// Mitsubishi GX Works2 project: BookEX6_44 Clock   PLC: Q13UDV

// global labels: Global
VAR_GLOBAL
  bVar0 AT M5000 : BOOL;
  abArray0 AT M5010 : ARRAY [0..49] OF BOOL;
  sStr0 AT D5000 : STRING[199];
  sStr1 AT D5100 : STRING[199];
  sStr2 AT D5200 : STRING[199];
  sStr3 AT D5300 : STRING[199];
  sStr4 AT D5400 : STRING[199];
  sStr5 AT D5500 : STRING[199];
  sStr6 AT D5600 : STRING[199];
  sStr7 AT D5700 : STRING[199];
  sStr8 AT D5800 : STRING[199];
  sStr9 AT D5900 : STRING[199];
  iVar0 AT D4500 : INT;
  iVar1 AT D4501 : INT;
  iVar2 AT D4502 : INT;
  iVar3 AT D4503 : INT;
  iVar4 AT D4504 : INT;
  iVar5 AT D4505 : INT;
  iVar6 AT D4506 : INT;
  iVar7 AT D4507 : INT;
  iVar8 AT D4508 : INT;
  iVar9 AT D4509 : INT;
  dVar0 AT D4510 : DINT;
  dVar1 AT D4512 : DINT;
  dVar2 AT D4514 : DINT;
  dVar3 AT D4516 : DINT;
  dVar4 AT D4518 : DINT;
  dVar5 AT D4520 : DINT;
  dVar6 AT D4522 : DINT;
  dVar7 AT D4524 : DINT;
  dVar8 AT D4526 : DINT;
  dVar9 AT D4528 : DINT;
  wVar0 AT D4530 : WORD;
  wVar1 AT D4531 : WORD;
  wVar2 AT D4532 : WORD;
  wVar3 AT D4533 : WORD;
  wVar4 AT D4534 : WORD;
  wVar5 AT D4535 : WORD;
  wVar6 AT D4536 : WORD;
  wVar7 AT D4537 : WORD;
  wVar8 AT D4538 : WORD;
  wVar9 AT D4539 : WORD;
  dwVar0 AT D4540 : DWORD;
  dwVar1 AT D4542 : DWORD;
  dwVar2 AT D4544 : DWORD;
  dwVar3 AT D4546 : DWORD;
  dwVar4 AT D4548 : DWORD;
  dwVar5 AT D4550 : DWORD;
  dwVar6 AT D4552 : DWORD;
  dwVar7 AT D4554 : DWORD;
  dwVar8 AT D4556 : DWORD;
  dwVar9 AT D4558 : DWORD;
  fsVar0 AT D4560 : REAL;
  fsVar1 AT D4562 : REAL;
  fsVar2 AT D4564 : REAL;
  fsVar3 AT D4566 : REAL;
  fsVar4 AT D4568 : REAL;
  fsVar5 AT D4570 : REAL;
  fsVar6 AT D4572 : REAL;
  fsVar7 AT D4574 : REAL;
  fsVar8 AT D4576 : REAL;
  fsVar9 AT D4578 : REAL;
  fdVar0 AT D4580 : LREAL;
  tTime0 AT D4620 : TIME;
  tTime1 AT D4622 : TIME;
  tTime2 AT D4624 : TIME;
  tTime3 AT D4626 : TIME;
  tTime4 AT D4628 : TIME;
  tTime5 AT D4630 : TIME;
  tTime6 AT D4632 : TIME;
  tTime7 AT D4634 : TIME;
  tTime8 AT D4636 : TIME;
  tTime9 AT D4638 : TIME;
  tTime10 AT D4640 : TIME;
  bVar1 AT M5001 : BOOL;
  bVar2 AT M5002 : BOOL;
  bVar3 AT M5003 : BOOL;
  bVar4 AT M5004 : BOOL;
  bVar5 AT M5005 : BOOL;
  bVar6 AT M5006 : BOOL;
  bVar7 AT M5007 : BOOL;
  bVar8 AT M5008 : BOOL;
  bVar9 AT M5009 : BOOL;
  abArray1 AT M5060 : ARRAY [0..49] OF BOOL;
  abArray2 AT M5110 : ARRAY [0..49] OF BOOL;
  abArray3 AT M5160 : ARRAY [0..49] OF BOOL;
  abArray4 AT M5210 : ARRAY [0..49] OF BOOL;
  abArray5 AT M5260 : ARRAY [0..49] OF BOOL;
  abArray6 AT M5310 : ARRAY [0..49] OF BOOL;
  abArray7 AT M5360 : ARRAY [0..49] OF BOOL;
  abArray8 AT M5410 : ARRAY [0..49] OF BOOL;
  abArray9 AT M5460 : ARRAY [0..49] OF BOOL;
  fdVar1 AT D4584 : LREAL;
  fdVar2 AT D4588 : LREAL;
  fdVar3 AT D4592 : LREAL;
  fdVar4 AT D4596 : LREAL;
  fdVar5 AT D4600 : LREAL;
  fdVar6 AT D4604 : LREAL;
  fdVar7 AT D4608 : LREAL;
  fdVar8 AT D4612 : LREAL;
  fdVar9 AT D4616 : LREAL;
  afsPen0 AT D2000 : ARRAY [0..499] OF REAL;
  afsPen1 AT D3000 : ARRAY [0..499] OF REAL;
  adwD10 AT D10 : ARRAY [0..9] OF DWORD;
  awD10 AT D10 : ARRAY [0..19] OF WORD;
  abM10 AT M10 : ARRAY [0..19] OF BOOL;
  bDown AT M50 : BOOL;
  bUp AT M51 : BOOL;
  bResult AT M325 : ARRAY [0..2] OF BOOL;
  bResultCMP1 AT M328 : ARRAY [0..2] OF BOOL;
  bResultCMP2 AT M331 : ARRAY [0..2] OF BOOL;
  bResultCP1 AT M334 : ARRAY [0..2] OF BOOL;
  bResultCP2 AT M337 : ARRAY [0..2] OF BOOL;
  aiClock AT D40 : ARRAY [0..6] OF INT;
  aiClock1 AT D40 : ARRAY [0..7] OF INT;
  aiClock2 AT D40 : ARRAY [0..5] OF INT;
  iInYear AT D48 : INT;
  iInMonth AT D49 : INT;
  asDay AT D100 : ARRAY [0..49] OF STRING[3] := [50('')];
  aiLowDate AT D330 : ARRAY [0..5] OF INT;
  aiLowTime AT D333 : ARRAY [0..2] OF INT;
  aiHighDate AT D340 : ARRAY [0..5] OF INT;
  aiHighTime AT D343 : ARRAY [0..2] OF INT;
  aiChkDate AT D350 : ARRAY [0..5] OF INT;
  aiChkTime AT D353 : ARRAY [0..2] OF INT;
  aiCnvTime AT D360 : ARRAY [0..2] OF INT;
  dCnvSec AT D363 : DINT;
END_VAR
// user libraries (not included): HMI

FUNCTION_BLOCK Calendar
VAR_INPUT
  i_Year : INT;
  i_Month : INT;
END_VAR
VAR
  oldYear : INT;
  oldMonth : INT;
  Days : INT;
  GetLastDay_1 : GetLastDay;
  ix : INT;
  iy : INT;
  iz : INT;
  sTemp : STRING[9];
  sForm : DINT;
  GetDayOfWeek_1 : GetDayOfWeek;
END_VAR
;

IF (oldMonth = i_Month) AND (oldYear = i_Year) THEN
	RETURN;
END_IF;

GetLastDay_1(bEN:= TRUE, iYear:= i_Year, iMonth:= i_Month );
Days := GetLastDay_1.o_LastDay;
GetDayOfWeek_1(bEN:=TRUE,iYear:= i_Year, iMonth:= i_Month, iDay:= 1);
iy :=  GetDayOfWeek_1.o_DayWeek;
iz := iy + Days;
sForm := 3;

FOR ix := 0 TO 41 DO 
	IF ( ix >= iy ) AND ( ix < iz) THEN
		STR(TRUE, sForm, ix-iy+1, sTemp);
		sTemp := DELETE(sTemp, 1, 1); 
	ELSE
		sTemp := '';
	END_IF;	
	asDay[ix] := sTemp;
END_FOR;

oldMonth := i_Month;
oldYear := i_Year;
END_FUNCTION_BLOCK

FUNCTION_BLOCK CmpDateZone
VAR_INPUT
  bEN : BOOL;
END_VAR
VAR_OUTPUT
  bENO : BOOL;
END_VAR
VAR_INPUT
  LowerLimit : ARRAY [0..5] OF INT;
  UpperLimit : ARRAY [0..5] OF INT;
  CheckDate : ARRAY [0..5] OF INT;
END_VAR
VAR_OUTPUT
  bLower : BOOL;
  bInner : BOOL;
  bUpper : BOOL;
END_VAR
VAR
  dLLimit : DINT;
  dULimit : DINT;
  dChkDate : DINT;
  bChkBit : ARRAY [0..2] OF BOOL;
  bChkData1 : BOOL;
  bChkData2 : BOOL;
  bChkData3 : BOOL;
END_VAR

bENO 	:= bEN;
bChkBit[0]	:= FALSE;
bChkBit[1]	:= FALSE;
bChkBit[2]	:= FALSE;
bChkData1 := (CheckDate[0]<2000) OR (CheckDate[0]>2067) 
  	OR (CheckDate[1]=0) OR (CheckDate[1]>12) 
  	OR (CheckDate[2]=0) OR (CheckDate[2]>31)  
  	OR (CheckDate[3]>23) OR (CheckDate[4]>59) OR (CheckDate[5]>59);
bChkData2 := (LowerLimit[0]<2000) OR (LowerLimit[0]>2067) 
  	OR (LowerLimit[1]=0) OR (LowerLimit[1]>12) 
  	OR (LowerLimit[2]=0) OR (LowerLimit[2]>31)  
  	OR (LowerLimit[3]>23) OR (LowerLimit[4]>59) OR (LowerLimit[5]>59);
bChkData3 := (UpperLimit[0]<2000) OR (UpperLimit[0]>2067) 
  	OR (UpperLimit[1]=0) OR (UpperLimit[1]>12) 
  	OR (UpperLimit[2]=0) OR (UpperLimit[2]>31)  
  	OR (UpperLimit[3]>23) OR (UpperLimit[4]>59) OR (UpperLimit[5]>59);
  		  		 
IF NOT bEN OR bChkData1 OR bChkData2 OR bChkData3 THEN
	RETURN;
END_IF; 
  
dLLimit := newDATE2SEC(LowerLimit[0], LowerLimit[1], LowerLimit[2], LowerLimit[3], LowerLimit[4], LowerLimit[5]);
dULimit := newDATE2SEC(UpperLimit[0], UpperLimit[1],UpperLimit[2],UpperLimit[3],UpperLimit[4],UpperLimit[5]); 
dChkDate := newDATE2SEC(CheckDate[0], CheckDate[1],CheckDate[2],CheckDate[3],CheckDate[4],CheckDate[5]);
IF dLLimit > dChkDate THEN
	bChkBit[0] := TRUE;
ELSIF dULimit < dChkDate THEN	
	bChkBit[2] := TRUE;
ELSE
	bChkBit[1] := TRUE;
END_IF;
bLower	:= bChkBit[0];
bUpper	:= bChkBit[2];
bInner	:= bChkBit[1];
END_FUNCTION_BLOCK

FUNCTION_BLOCK GetDayOfWeek
VAR_INPUT
  bEN : BOOL;
END_VAR
VAR_OUTPUT
  bENO : BOOL;
END_VAR
VAR_INPUT
  iYear : INT;
END_VAR
VAR_OUTPUT
  o_DayWeek : INT;
END_VAR
VAR
  Result : INT;
END_VAR
VAR_INPUT
  iMonth : INT;
  iDay : INT;
END_VAR
VAR
  iY : INT;
  iC : INT;
  iM : INT;
  iYear2 : INT;
END_VAR

bENO 	:= bEN;
IF NOT bEN THEN
	RETURN;
END_IF;
IF iMonth <= 2 THEN
	iYear2 := iYear - 1;
	iM := iMonth + 12;
ELSE
	iYear2 := iYear;
	iM := iMonth;
END_IF;
iC := iYear2 / 100; 
iY := iYear2 MOD 100;
Result := ( (21*iC)/4 +(5* iY)/4 + (13 * (iM+1)) / 5 +iDay - 1) MOD 7; 
o_DayWeek := Result;
END_FUNCTION_BLOCK

FUNCTION_BLOCK GetLastDay
VAR_INPUT
  bEN : BOOL;
END_VAR
VAR_OUTPUT
  bENO : BOOL;
END_VAR
VAR_INPUT
  iYear : INT;
END_VAR
VAR_OUTPUT
  o_LastDay : INT;
END_VAR
VAR
  Result : INT;
END_VAR
VAR_INPUT
  iMonth : INT;
END_VAR
VAR
  bLeap : BOOL;
END_VAR

bENO 	:= bEN;
IF NOT bEN THEN
	RETURN;
END_IF; 

bLeap := LeapYear(iYear);
CASE iMonth OF
	1 : Result	:= 31;
	2 : IF bLeap THEN Result := 29; ELSE Result	:= 28; END_IF;
	3 : Result	:= 31;
	4 : Result	:= 30;
	5 : Result	:= 31;
	6 : Result	:= 30;
	7 : Result	:= 31;
	8 : Result	:= 31;
	9 : Result	:= 30;
	10 : Result	:= 31;
	11 : Result	:= 30;
	12 : Result	:= 31;
END_CASE;	
o_LastDay := Result;
END_FUNCTION_BLOCK

FUNCTION_BLOCK HourMeter
VAR_INPUT
  bEN : BOOL;
END_VAR
VAR_OUTPUT
  bENO : BOOL;
END_VAR
VAR_INPUT
  iHour : INT;
  iCurrHour : INT;
  iCurrSec : INT;
END_VAR
VAR_OUTPUT
  etHour : INT;
  etSec : INT;
  bOut : BOOL;
END_VAR
VAR
  tmpHour : INT;
  tmpSec : INT;
  R_TRIG_1 : R_TRIG;
END_VAR

bENO 	:= bEN;
IF LDP(TRUE, bEN) THEN
	tmpHour	:= iCurrHour;
	tmpSec	:= iCurrSec;
	bOut	:= FALSE;
END_IF;
IF NOT bEN THEN
	RETURN;
END_IF; 


IF LDP(TRUE, SM412) THEN
	tmpSec	:= tmpSec+1;
	IF tmpSec > 3599 THEN
		tmpSec	:= 0;
		tmpHour	:= tmpHour+1;
	END_IF;
	IF tmpHour = iHour THEN
		bOut	:= TRUE;
	END_IF;
END_IF;

etHour	:= tmpHour;
etSec	:= tmpSec;
END_FUNCTION_BLOCK

FUNCTION LeapYear
VAR
  bLeap4 : BOOL;
  bLeap100 : BOOL;
  bLeap400 : BOOL;
END_VAR
VAR_INPUT
  i_Year : INT;
END_VAR
VAR
  bLeap : BOOL;
END_VAR
;
bLeap := FALSE;
IF (i_Year MOD 4) = 0 THEN bLeap4 := TRUE; ELSE bLeap4 := FALSE; END_IF;
IF (i_Year MOD 100) = 0 THEN bLeap100 := TRUE; ELSE bLeap100 := FALSE; END_IF;
IF (i_Year MOD 400) = 0 THEN bLeap400 := TRUE; ELSE bLeap400 := FALSE; END_IF;
IF (bLeap4 AND NOT bLeap100) OR bLeap400 THEN bLeap := TRUE; END_IF;
LeapYear := bLeap;
END_FUNCTION

FUNCTION newDATE2SEC
VAR_INPUT
  i_Year : INT;
  i_Month : INT;
  i_Day : INT;
  i_Hour : INT;
  i_Min : INT;
  i_Sec : INT;
END_VAR
VAR
  ix : INT;
  dDay : DINT;
  diDay : DINT;
END_VAR
;
IF i_Year  < 2000  OR i_Year > 2067 THEN 
	newDATE2SEC := 0;
	RETURN;
END_IF; 
dDay := 0;
IF i_Year > 2000 THEN
	FOR ix := 2000 TO i_Year-1 DO 
		IF LeapYear(ix) THEN
			dDay := dDay + 366;
		ELSE
			dDay := dDay + 365;
		END_IF;
	END_FOR;
END_IF;
diDay := INT_TO_DINT(i_Day-1);
CASE i_Month OF
	1 : 	dDay := dDay + diDay;
	2 :	dDay := dDay + 31 + diDay;
	3 : 	dDay := dDay + 31 + 28 + diDay;
	4 : 	dDay := dDay + 31 + 28 + 31 + diDay;
	5 : 	dDay := dDay + 31 + 28 + 31 + 30 + diDay;
	6 : 	dDay := dDay + 31 + 28 + 31 + 30 + 31 + diDay;
	7 : 	dDay := dDay + 31 + 28 + 31 + 30 + 31 + 30 + diDay;
	8 : 	dDay := dDay + 31 + 28 + 31 + 30 + 31 + 30 + 31 + diDay;
	9 : 	dDay := dDay + 31 + 28 + 31 + 30 + 31 + 30 + 31 + 31 + diDay;
	10 : 	dDay := dDay + 31 + 28 + 31 + 30 + 31 + 30 + 31 + 31 + 30 + diDay;
	11 : 	dDay := dDay + 31 + 28 + 31 + 30 + 31 + 30 + 31 + 31 + 30 + 31 + diDay;
	12 : 	dDay := dDay + 31 + 28 + 31 + 30 + 31 + 30 + 31 + 31 + 30 + 31 + 30 + diDay;
ELSE
	dDay := 0;
END_CASE;
IF i_Month > 2 AND LeapYear(i_Year) THEN dDay := dDay + 1; END_IF;
newDATE2SEC := dDay * 24* 60 * 60 + INT_TO_DINT(i_Hour) * 60 * 60 + INT_TO_DINT(i_Min) * 60 + INT_TO_DINT(i_Sec);
END_FUNCTION

FUNCTION_BLOCK sysDateTime
VAR_OUTPUT
  Secs : INT;
  Mins : INT;
  Hours : INT;
  Day : INT;
  Month : INT;
  Year : INT;
END_VAR
VAR
  Temp2 : WORD;
  Temp1 : WORD;
  fbTimer : TON;
  SeqGet : INT;
END_VAR
(* PLC의 realtime clock data를 읽는다 *)
SM213 := TRUE;
(* Year *)
Temp1 := SHR(INT_TO_WORD(SD210) AND 16#FF00, 8);
Temp2 := INT_TO_WORD(SD213) AND 16#FF00;
BIN(TRUE, Temp1 OR Temp2, Year);
(* Month *)
Temp1 := INT_TO_WORD(SD210) AND 16#00FF;
BIN(TRUE, Temp1, Month);
(* Day *)
Temp1 := SHR(INT_TO_WORD(SD211) AND 16#FF00, 8);
BIN(TRUE, Temp1, Day);
(* Hour *)
Temp1 := INT_TO_WORD(SD211) AND 16#00FF;
BIN(TRUE, Temp1, Hours);
(* Minute *)
Temp1 := SHR(INT_TO_WORD(SD212) AND 16#FF00, 8);
BIN(TRUE, Temp1, Mins);
(* Second *)
Temp1 := INT_TO_WORD(SD212) AND 16#00FF;
BIN(TRUE, Temp1, Secs);
END_FUNCTION_BLOCK

PROGRAM ExCalendar
VAR
  Calendar_1 : Calendar;
  aiMin : ARRAY [0..1] OF INT;
  aiSec : ARRAY [0..1] OF INT;
  aiHour : ARRAY [0..1] OF INT;
END_VAR
(* structured ladder/FBD written out as ST: instructions are called as NAME(EN, inputs, outputs); _pN, _eN, _tN stand for wires *)
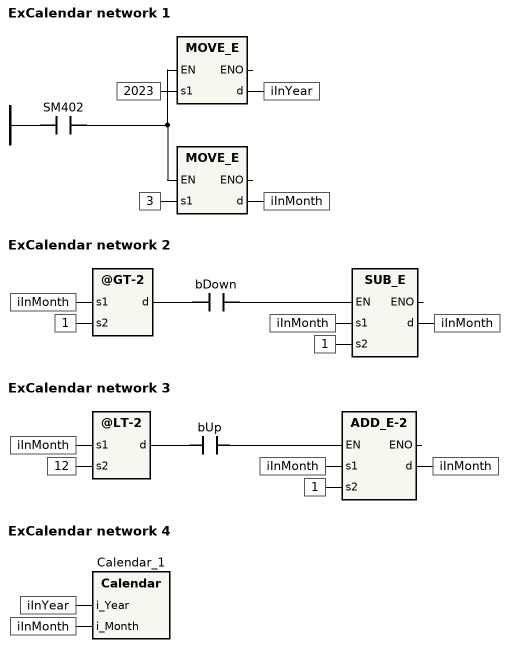
(* network 1 *)
MOVE_E(SM402, 2023, iInYear);
MOVE_E(SM402, 3, iInMonth);
(* network 2 *)
SUB_E(@GT-2(iInMonth, 1) AND bDown, iInMonth, 1, iInMonth);
(* network 3 *)
ADD_E(@LT-2(iInMonth, 12) AND bUp, iInMonth, 1, iInMonth);
(* network 4 *)
Calendar_1(i_Year := iInYear, i_Month := iInMonth);
END_PROGRAM

PROGRAM ExClcok
VAR
  Calendar_1 : Calendar;
  aiMin : ARRAY [0..1] OF INT;
  aiSec : ARRAY [0..1] OF INT;
  aiHour : ARRAY [0..1] OF INT;
END_VAR
(* structured ladder/FBD written out as ST: instructions are called as NAME(EN, inputs, outputs); _pN, _eN, _tN stand for wires *)
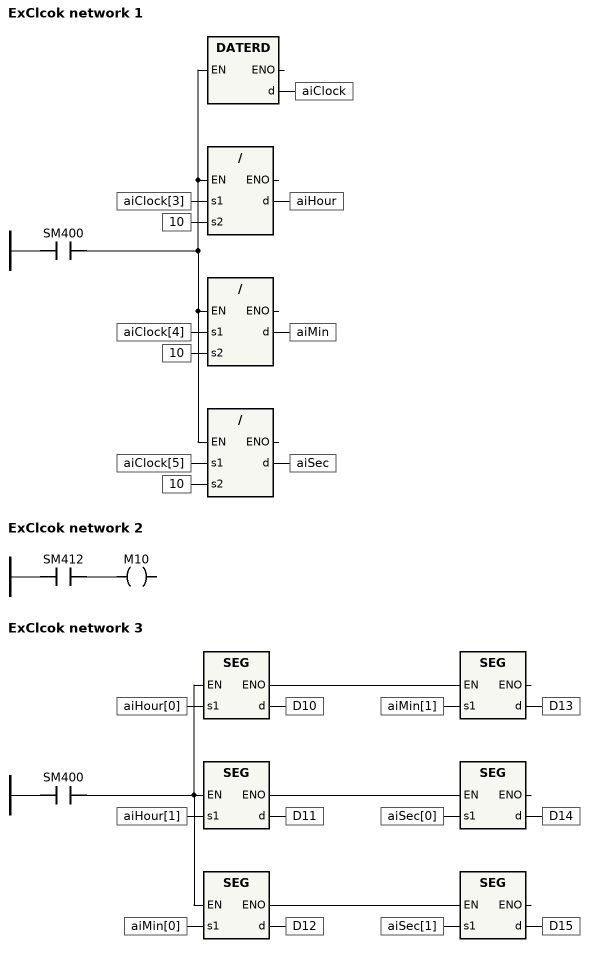
(* network 1 *)
DATERD(SM400, aiClock);
/(SM400, aiClock[3], 10, aiHour);
/(SM400, aiClock[4], 10, aiMin);
/(SM400, aiClock[5], 10, aiSec);
(* network 2 *)
M10 := SM412;
(* network 3 *)
_e1 := SEG(SM400, aiHour[0], D10);
SEG(_e1, aiMin[1], D13);
_e2 := SEG(SM400, aiHour[1], D11);
SEG(_e2, aiSec[0], D14);
_e3 := SEG(SM400, aiMin[0], D12);
SEG(_e3, aiSec[1], D15);
END_PROGRAM

PROGRAM ExDATE2SEC
VAR
  aiDate : ARRAY [0..5] OF INT;
END_VAR
(* structured ladder/FBD written out as ST: instructions are called as NAME(EN, inputs, outputs); _pN, _eN, _tN stand for wires *)
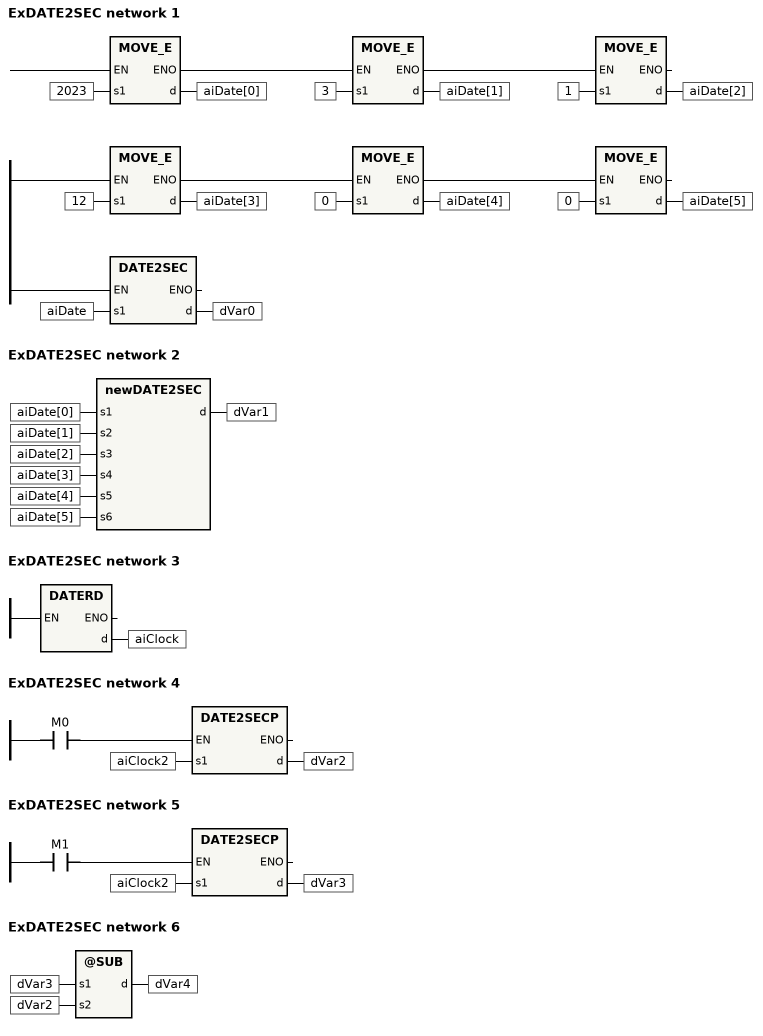
(* network 1 *)
_e1 := MOVE_E(TRUE, 2023, aiDate[0]);
_e2 := MOVE_E(_e1, 3, aiDate[1]);
MOVE_E(_e2, 1, aiDate[2]);
_e3 := MOVE_E(TRUE, 12, aiDate[3]);
_e4 := MOVE_E(_e3, 0, aiDate[4]);
MOVE_E(_e4, 0, aiDate[5]);
DATE2SEC(TRUE, aiDate, dVar0);
(* network 2 *)
dVar1 := newDATE2SEC(aiDate[0], aiDate[1], aiDate[2], aiDate[3], aiDate[4], aiDate[5]);
(* network 3 *)
DATERD(TRUE, aiClock);
(* network 4 *)
DATE2SECP(M0, aiClock2, dVar2);
(* network 5 *)
DATE2SECP(M1, aiClock2, dVar3);
(* network 6 *)
dVar4 := @SUB(dVar3, dVar2);
END_PROGRAM

PROGRAM ExDateMinus
VAR
  Mov4INT_3 : Mov4INT;
  Mov4INT_4 : Mov4INT;
  aiTime1 : ARRAY [0..2] OF INT;
  aiTime2 : ARRAY [0..2] OF INT;
  aiTime3 : ARRAY [0..2] OF INT;
  Mov4INT_1 : Mov4INT;
END_VAR
(* structured ladder/FBD written out as ST: instructions are called as NAME(EN, inputs, outputs); _pN, _eN, _tN stand for wires *)
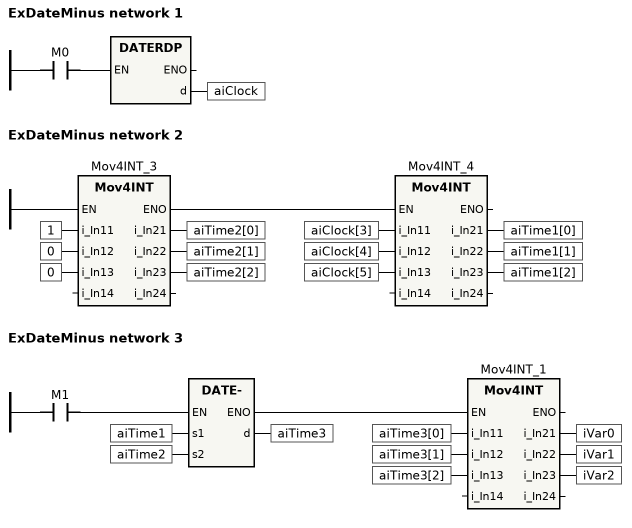
(* network 1 *)
DATERDP(M0, aiClock);
(* network 2 *)
Mov4INT_3(EN := TRUE, i_In11 := 1, i_In12 := 0, i_In13 := 0, i_In21 => aiTime2[0], i_In22 => aiTime2[1], i_In23 => aiTime2[2]);
Mov4INT_4(EN := Mov4INT_3.ENO, i_In11 := aiClock[3], i_In12 := aiClock[4], i_In13 := aiClock[5], i_In21 => aiTime1[0], i_In22 => aiTime1[1], i_In23 => aiTime1[2]);
(* network 3 *)
_e1 := DATE-(M1, aiTime1, aiTime2, aiTime3);
Mov4INT_1(EN := _e1, i_In11 := aiTime3[0], i_In12 := aiTime3[1], i_In13 := aiTime3[2], i_In21 => iVar0, i_In22 => iVar1, i_In23 => iVar2);
END_PROGRAM

PROGRAM ExDatePlus
VAR
  Mov4INT_3 : Mov4INT;
  Mov4INT_4 : Mov4INT;
  aiTime1 : ARRAY [0..2] OF INT;
  aiTime2 : ARRAY [0..2] OF INT;
  aiTime3 : ARRAY [0..2] OF INT;
  Mov4INT_1 : Mov4INT;
END_VAR
(* structured ladder/FBD written out as ST: instructions are called as NAME(EN, inputs, outputs); _pN, _eN, _tN stand for wires *)
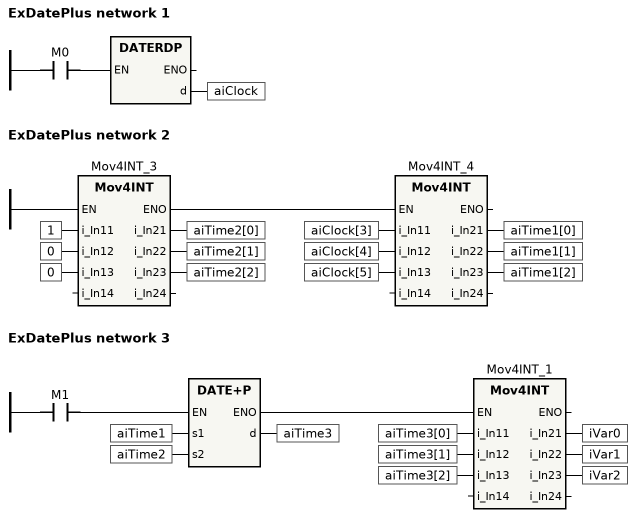
(* network 1 *)
DATERDP(M0, aiClock);
(* network 2 *)
Mov4INT_3(EN := TRUE, i_In11 := 1, i_In12 := 0, i_In13 := 0, i_In21 => aiTime2[0], i_In22 => aiTime2[1], i_In23 => aiTime2[2]);
Mov4INT_4(EN := Mov4INT_3.ENO, i_In11 := aiClock[3], i_In12 := aiClock[4], i_In13 := aiClock[5], i_In21 => aiTime1[0], i_In22 => aiTime1[1], i_In23 => aiTime1[2]);
(* network 3 *)
_e1 := DATE+P(M1, aiTime1, aiTime2, aiTime3);
Mov4INT_1(EN := _e1, i_In11 := aiTime3[0], i_In12 := aiTime3[1], i_In13 := aiTime3[2], i_In21 => iVar0, i_In22 => iVar1, i_In23 => iVar2);
END_PROGRAM

PROGRAM ExDATERD
VAR
  wBCD1 : WORD;
  wBCD2 : WORD;
  wBCD3 : WORD;
  wBCD4 : WORD;
  wBCD5 : WORD;
  wBCD6 : WORD;
  wBCD7 : WORD;
  wBCD8 : WORD;
  iTime1 : INT;
  iTime2 : INT;
  iTime3 : INT;
  iTime4 : INT;
  iTime5 : INT;
  iTime6 : INT;
  iTime7 : INT;
  iTime8 : INT;
  sysDateTime_1 : sysDateTime;
  Mov8INT2BCD_1 : Mov8INT2BCD;
END_VAR
(* structured ladder/FBD written out as ST: instructions are called as NAME(EN, inputs, outputs); _pN, _eN, _tN stand for wires *)
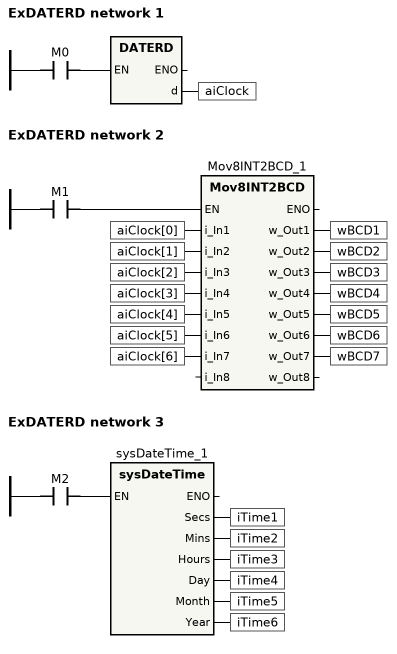
(* network 1 *)
DATERD(M0, aiClock);
(* network 2 *)
Mov8INT2BCD_1(EN := M1, i_In1 := aiClock[0], i_In2 := aiClock[1], i_In3 := aiClock[2], i_In4 := aiClock[3], i_In5 := aiClock[4], i_In6 := aiClock[5], i_In7 := aiClock[6], w_Out1 => wBCD1, w_Out2 => wBCD2, w_Out3 => wBCD3, w_Out4 => wBCD4, w_Out5 => wBCD5, w_Out6 => wBCD6, w_Out7 => wBCD7);
(* network 3 *)
sysDateTime_1(EN := M2, Secs => iTime1, Mins => iTime2, Hours => iTime3, Day => iTime4, Month => iTime5, Year => iTime6);
END_PROGRAM

PROGRAM ExDateWR
VAR
  acVar0 : ARRAY [0..6] OF INT;
END_VAR
(* structured ladder/FBD written out as ST: instructions are called as NAME(EN, inputs, outputs); _pN, _eN, _tN stand for wires *)
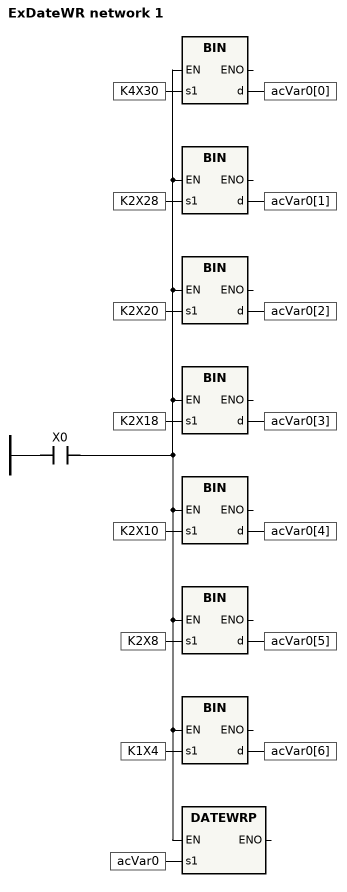
(* network 1 *)
BIN(X0, K4X30, acVar0[0]);
BIN(X0, K2X28, acVar0[1]);
BIN(X0, K2X20, acVar0[2]);
BIN(X0, K2X18, acVar0[3]);
BIN(X0, K2X10, acVar0[4]);
BIN(X0, K2X8, acVar0[5]);
BIN(X0, K1X4, acVar0[6]);
DATEWRP(X0, acVar0);
END_PROGRAM

PROGRAM ExGetLastDay
VAR
  GetLastDay_1 : GetLastDay;
  GetLastDay_2 : GetLastDay;
  GetLastDay_3 : GetLastDay;
  GetLastDay_4 : GetLastDay;
  GetLastDay_5 : GetLastDay;
  GetLastDay_6 : GetLastDay;
END_VAR
(* structured ladder/FBD written out as ST: instructions are called as NAME(EN, inputs, outputs); _pN, _eN, _tN stand for wires *)
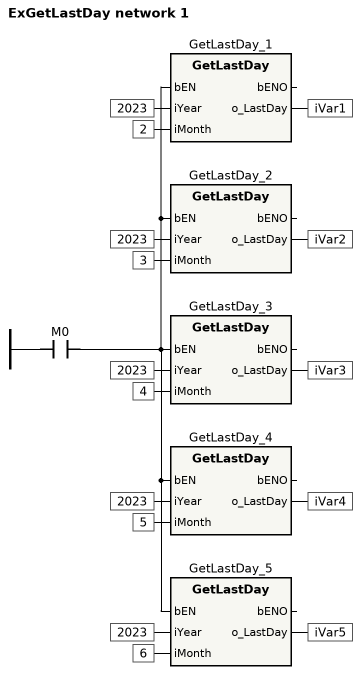
(* network 1 *)
GetLastDay_1(bEN := M0, iYear := 2023, iMonth := 2, o_LastDay => iVar1);
GetLastDay_2(bEN := M0, iYear := 2023, iMonth := 3, o_LastDay => iVar2);
GetLastDay_3(bEN := M0, iYear := 2023, iMonth := 4, o_LastDay => iVar3);
GetLastDay_4(bEN := M0, iYear := 2023, iMonth := 5, o_LastDay => iVar4);
GetLastDay_5(bEN := M0, iYear := 2023, iMonth := 6, o_LastDay => iVar5);
END_PROGRAM

PROGRAM ExHOUR
VAR
  aiVar3 : ARRAY [0..2] OF INT;
  iHourData : INT;
  iSecData : INT;
  aiVar4 : ARRAY [0..2] OF INT;
END_VAR
(* structured ladder/FBD written out as ST: instructions are called as NAME(EN, inputs, outputs); _pN, _eN, _tN stand for wires *)
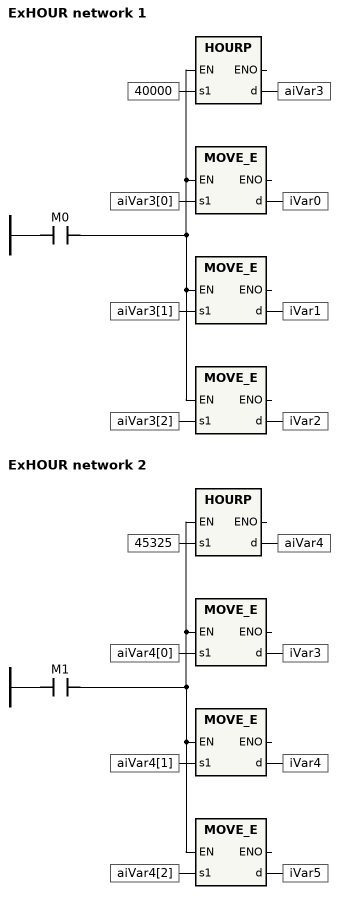
(* network 1 *)
HOURP(M0, 40000, aiVar3);
MOVE_E(M0, aiVar3[0], iVar0);
MOVE_E(M0, aiVar3[1], iVar1);
MOVE_E(M0, aiVar3[2], iVar2);
(* network 2 *)
HOURP(M1, 45325, aiVar4);
MOVE_E(M1, aiVar4[0], iVar3);
MOVE_E(M1, aiVar4[1], iVar4);
MOVE_E(M1, aiVar4[2], iVar5);
END_PROGRAM

PROGRAM ExHOURM
VAR
  iHourM : ARRAY [0..1] OF INT;
  iHourData : INT;
  iSecData : INT;
  iHourDM : ARRAY [0..2] OF INT;
  iHourDData : DINT;
  iSecDData : INT;
  HourMeter_1 : HourMeter;
  iHM_H : INT;
  iHM_S : INT;
END_VAR
(* structured ladder/FBD written out as ST: instructions are called as NAME(EN, inputs, outputs); _pN, _eN, _tN stand for wires *)
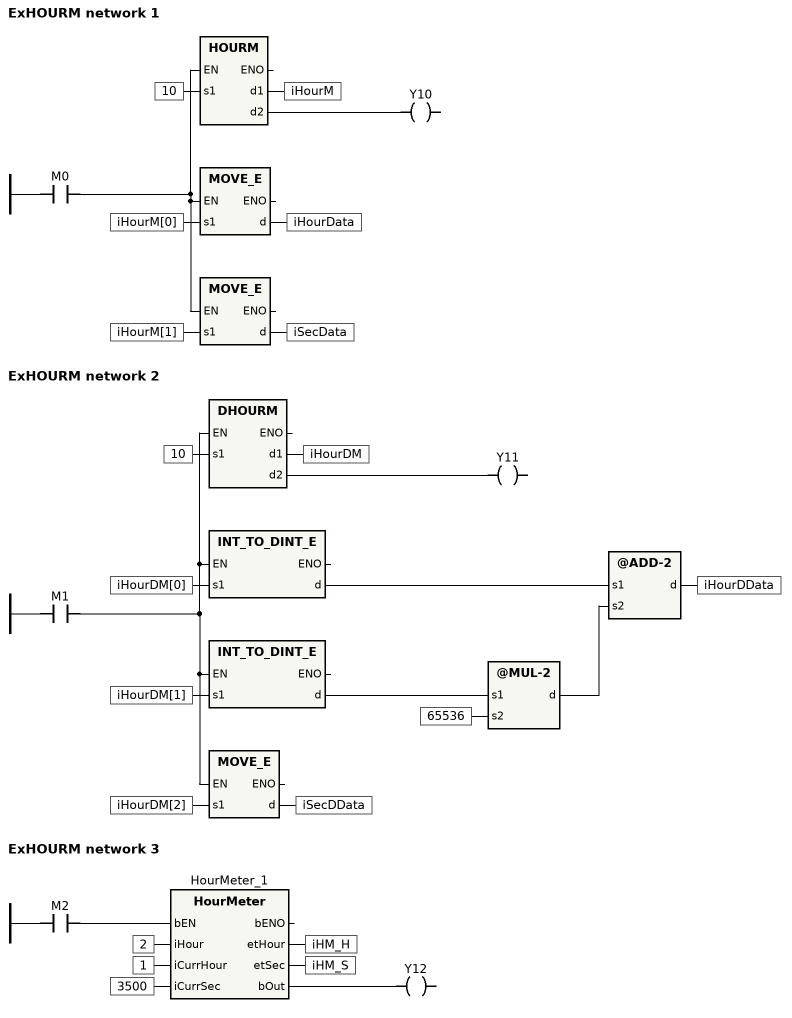
(* network 1 *)
HOURM(M0, 10, iHourM, _t1);
Y10 := _t1;
MOVE_E(M0, iHourM[0], iHourData);
MOVE_E(M0, iHourM[1], iSecData);
(* network 2 *)
DHOURM(M1, 10, iHourDM, _t1);
Y11 := _t1;
INT_TO_DINT_E(M1, iHourDM[0], _t2);
INT_TO_DINT_E(M1, iHourDM[1], _t3);
iHourDData := @ADD-2(_t2, @MUL-2(_t3, 65536));
MOVE_E(M1, iHourDM[2], iSecDData);
(* network 3 *)
HourMeter_1(bEN := M2, iHour := 2, iCurrHour := 1, iCurrSec := 3500, etHour => iHM_H, etSec => iHM_S);
Y12 := HourMeter_1.bOut;
END_PROGRAM

PROGRAM ExLDDT
VAR
  cmpDate : ARRAY [0..2] OF INT;
  Mov4INT_1 : Mov4INT;
  Mov4INT_2 : Mov4INT;
  Mov4INT_3 : Mov4INT;
  Mov4INT_4 : Mov4INT;
END_VAR
(* structured ladder/FBD written out as ST: instructions are called as NAME(EN, inputs, outputs); _pN, _eN, _tN stand for wires *)
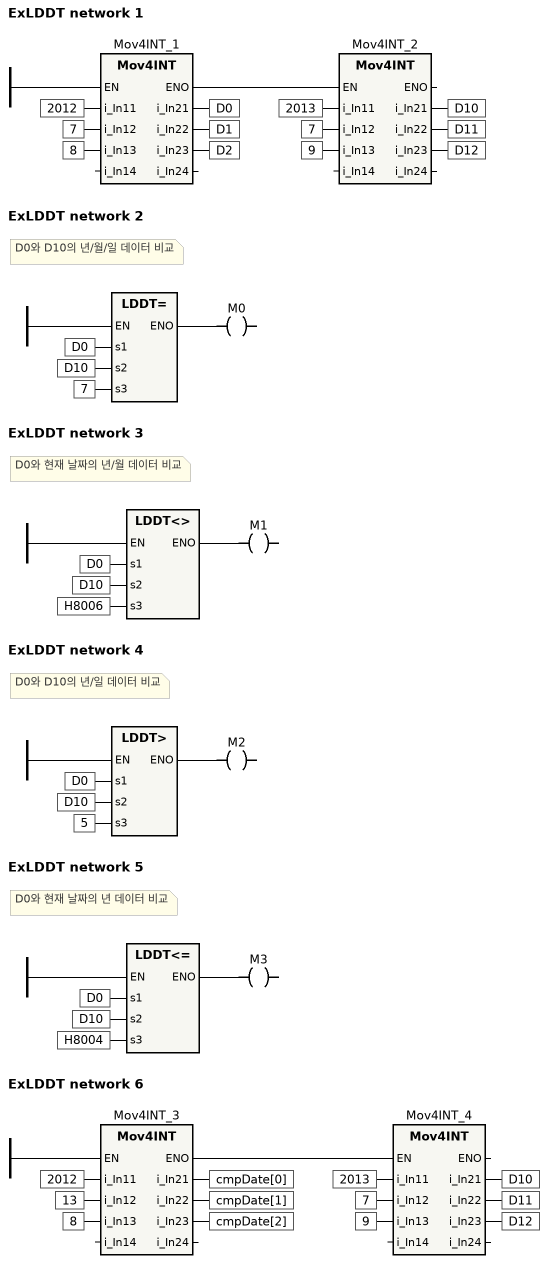
(* network 1 *)
Mov4INT_1(EN := TRUE, i_In11 := 2012, i_In12 := 7, i_In13 := 8, i_In21 => D0, i_In22 => D1, i_In23 => D2);
Mov4INT_2(EN := Mov4INT_1.ENO, i_In11 := 2013, i_In12 := 7, i_In13 := 9, i_In21 => D10, i_In22 => D11, i_In23 => D12);
(* network 2 *)
(* D0와 D10의 년/월/일 데이터 비교 *)
_e1 := LDDT=(TRUE, D0, D10, 7);
M0 := _e1;
(* network 3 *)
(* D0와 현재 날짜의 년/월 데이터 비교 *)
_e1 := LDDT<>(TRUE, D0, D10, H8006);
M1 := _e1;
(* network 4 *)
(* D0와 D10의 년/일 데이터 비교 *)
_e1 := LDDT>(TRUE, D0, D10, 5);
M2 := _e1;
(* network 5 *)
(* D0와 현재 날짜의 년 데이터 비교 *)
_e1 := LDDT<=(TRUE, D0, D10, H8004);
M3 := _e1;
(* network 6 *)
Mov4INT_3(EN := TRUE, i_In11 := 2012, i_In12 := 13, i_In13 := 8, i_In21 => cmpDate[0], i_In22 => cmpDate[1], i_In23 => cmpDate[2]);
Mov4INT_4(EN := Mov4INT_3.ENO, i_In11 := 2013, i_In12 := 7, i_In13 := 9, i_In21 => D10, i_In22 => D11, i_In23 => D12);
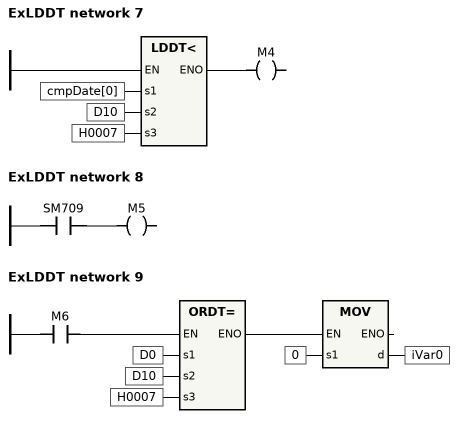
(* network 7 *)
_e1 := LDDT<(TRUE, cmpDate[0], D10, H0007);
M4 := _e1;
(* network 8 *)
M5 := SM709;
(* network 9 *)
_e1 := ORDT=(M6, D0, D10, H0007);
MOV(_e1, 0, iVar0);
END_PROGRAM

PROGRAM ExLDTM
VAR
  cmpTime : ARRAY [0..2] OF INT;
  Mov4INT_1 : Mov4INT;
  Mov4INT_2 : Mov4INT;
  Mov4INT_3 : Mov4INT;
  Mov4INT_4 : Mov4INT;
END_VAR
(* structured ladder/FBD written out as ST: instructions are called as NAME(EN, inputs, outputs); _pN, _eN, _tN stand for wires *)
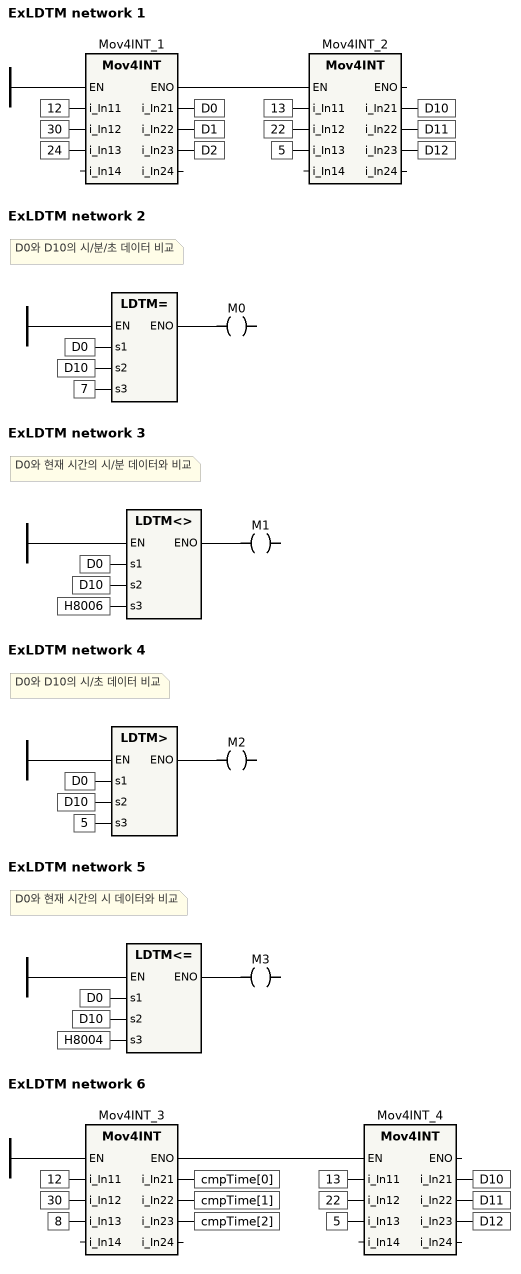
(* network 1 *)
Mov4INT_1(EN := TRUE, i_In11 := 12, i_In12 := 30, i_In13 := 24, i_In21 => D0, i_In22 => D1, i_In23 => D2);
Mov4INT_2(EN := Mov4INT_1.ENO, i_In11 := 13, i_In12 := 22, i_In13 := 5, i_In21 => D10, i_In22 => D11, i_In23 => D12);
(* network 2 *)
(* D0와 D10의 시/분/초 데이터 비교 *)
_e1 := LDTM=(TRUE, D0, D10, 7);
M0 := _e1;
(* network 3 *)
(* D0와 현재 시간의 시/분 데이터와 비교 *)
_e1 := LDTM<>(TRUE, D0, D10, H8006);
M1 := _e1;
(* network 4 *)
(* D0와 D10의 시/초 데이터 비교 *)
_e1 := LDTM>(TRUE, D0, D10, 5);
M2 := _e1;
(* network 5 *)
(* D0와 현재 시간의 시 데이터와 비교 *)
_e1 := LDTM<=(TRUE, D0, D10, H8004);
M3 := _e1;
(* network 6 *)
Mov4INT_3(EN := TRUE, i_In11 := 12, i_In12 := 30, i_In13 := 8, i_In21 => cmpTime[0], i_In22 => cmpTime[1], i_In23 => cmpTime[2]);
Mov4INT_4(EN := Mov4INT_3.ENO, i_In11 := 13, i_In12 := 22, i_In13 := 5, i_In21 => D10, i_In22 => D11, i_In23 => D12);
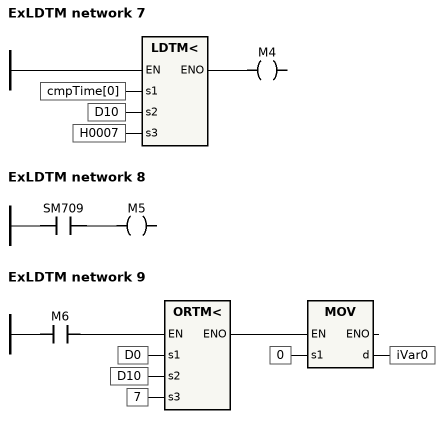
(* network 7 *)
_e1 := LDTM<(TRUE, cmpTime[0], D10, H0007);
M4 := _e1;
(* network 8 *)
M5 := SM709;
(* network 9 *)
_e1 := ORTM<(M6, D0, D10, 7);
MOV(_e1, 0, iVar0);
END_PROGRAM

PROGRAM ExSec2Date
VAR
  ix : INT;
  dSec : DINT;
  iy : INT;
  aiData : ARRAY [0..5] OF INT;
  aiData1 : ARRAY [0..6] OF INT;
END_VAR
;
IF iVar0  < 2000 THEN iy := 2000; ELSE iy := iVar0; END_IF; 
dSec := 0;
FOR ix := iy TO 2067 DO 
	IF LeapYear(ix) THEN
		dSec := dSec + 366;
	ELSE
		dSec := dSec + 365;
	END_IF;
END_FOR;
dSec := dSec * 24* 60 * 60;
dVar0 := dSec - 1;

aiData[0] := 2067;
aiData[1] := 12;
aiData[2] := 31;
aiData[3] := 23;
aiData[4] := 59;
aiData[5] := 59;
DATE2SEC(TRUE, aiData, dVar1);

dVar2 := 2145916799;
SEC2DATE(TRUE, dVar2, aiData1);
END_PROGRAM

PROGRAM ExSECOND
VAR
  acVar3 : ARRAY [0..2] OF INT;
END_VAR
(* structured ladder/FBD written out as ST: instructions are called as NAME(EN, inputs, outputs); _pN, _eN, _tN stand for wires *)
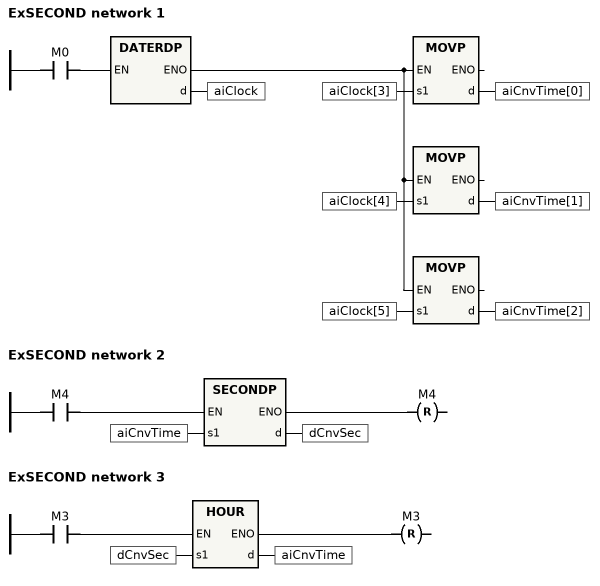
(* network 1 *)
_e1 := DATERDP(M0, aiClock);
MOVP(_e1, aiClock[3], aiCnvTime[0]);
MOVP(_e1, aiClock[4], aiCnvTime[1]);
MOVP(_e1, aiClock[5], aiCnvTime[2]);
(* network 2 *)
_e1 := SECONDP(M4, aiCnvTime, dCnvSec);
RST(_e1, M4);
(* network 3 *)
_e1 := HOUR(M3, dCnvSec, aiCnvTime);
RST(_e1, M3);
END_PROGRAM

PROGRAM ExTZCP
VAR
  abVar3 : ARRAY [0..2] OF BOOL;
  Mov4INT_1 : Mov4INT;
  aiTime1 : ARRAY [0..2] OF INT;
  aiTime2 : ARRAY [0..2] OF INT;
  aiTime3 : ARRAY [0..2] OF INT;
  Mov4INT_2 : Mov4INT;
  Mov4INT_3 : Mov4INT;
  Mov4INT_4 : Mov4INT;
  Mov4INT_5 : Mov4INT;
  Mov4INT_6 : Mov4INT;
  CmpDateZone_1 : CmpDateZone;
  Mov8INT_1 : Mov8INT;
  Mov8INT_2 : Mov8INT;
  Mov8INT_3 : Mov8INT;
  acVar3 : ARRAY [0..2] OF INT;
END_VAR
(* structured ladder/FBD written out as ST: instructions are called as NAME(EN, inputs, outputs); _pN, _eN, _tN stand for wires *)
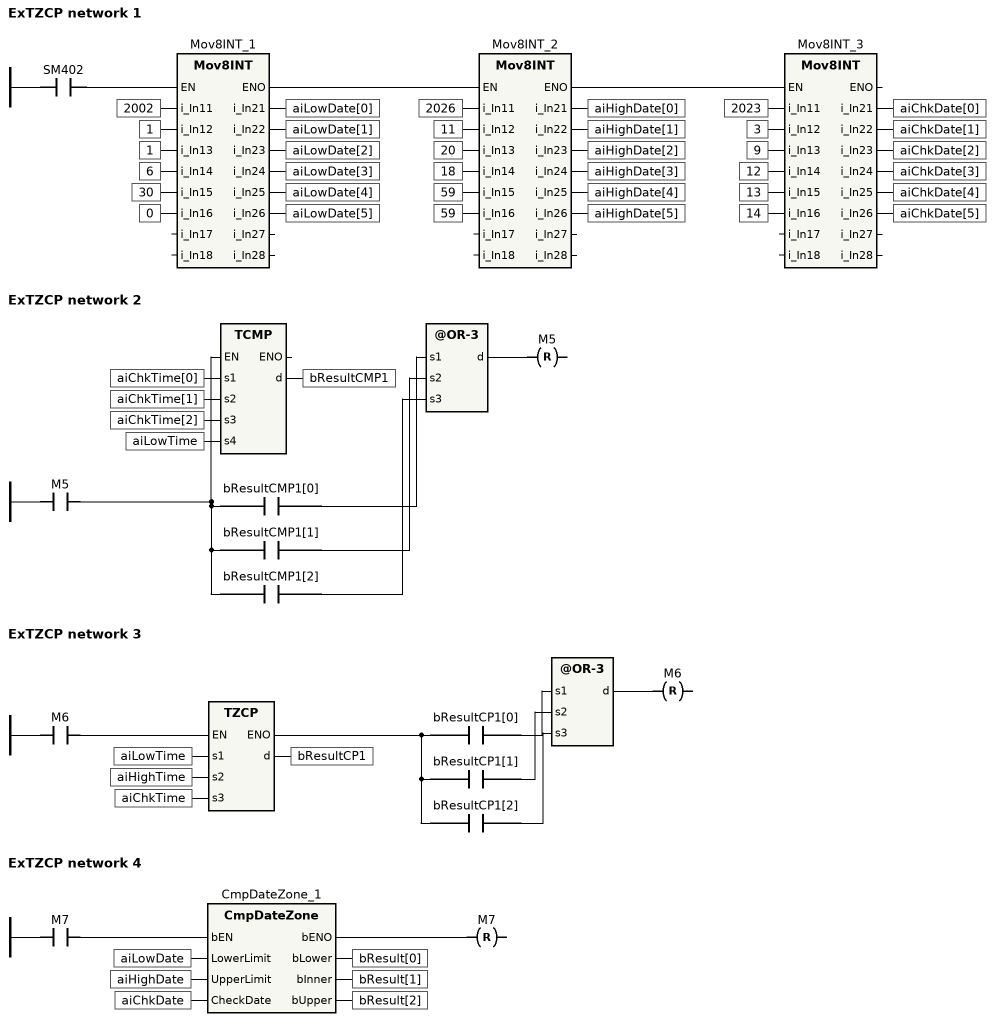
(* network 1 *)
Mov8INT_1(EN := SM402, i_In11 := 2002, i_In12 := 1, i_In13 := 1, i_In14 := 6, i_In15 := 30, i_In16 := 0, i_In21 => aiLowDate[0], i_In22 => aiLowDate[1], i_In23 => aiLowDate[2], i_In24 => aiLowDate[3], i_In25 => aiLowDate[4], i_In26 => aiLowDate[5]);
Mov8INT_2(EN := Mov8INT_1.ENO, i_In11 := 2026, i_In12 := 11, i_In13 := 20, i_In14 := 18, i_In15 := 59, i_In16 := 59, i_In21 => aiHighDate[0], i_In22 => aiHighDate[1], i_In23 => aiHighDate[2], i_In24 => aiHighDate[3], i_In25 => aiHighDate[4], i_In26 => aiHighDate[5]);
Mov8INT_3(EN := Mov8INT_2.ENO, i_In11 := 2023, i_In12 := 3, i_In13 := 9, i_In14 := 12, i_In15 := 13, i_In16 := 14, i_In21 => aiChkDate[0], i_In22 => aiChkDate[1], i_In23 => aiChkDate[2], i_In24 => aiChkDate[3], i_In25 => aiChkDate[4], i_In26 => aiChkDate[5]);
(* network 2 *)
TCMP(M5, aiChkTime[0], aiChkTime[1], aiChkTime[2], aiLowTime, bResultCMP1);
RST(@OR-3(M5 AND bResultCMP1[0], M5 AND bResultCMP1[1], M5 AND bResultCMP1[2]), M5);
(* network 3 *)
_e1 := TZCP(M6, aiLowTime, aiHighTime, aiChkTime, bResultCP1);
RST(@OR-3(_e1 AND bResultCP1[0], _e1 AND bResultCP1[1], _e1 AND bResultCP1[2]), M6);
(* network 4 *)
CmpDateZone_1(bEN := M7, LowerLimit := aiLowDate, UpperLimit := aiHighDate, CheckDate := aiChkDate, bLower => bResult[0], bInner => bResult[1], bUpper => bResult[2]);
RST(CmpDateZone_1.bENO, M7);
END_PROGRAM
